TYPE Kilogram : LREAL;
END_TYPE

(* stored: Version 1.1.0.1, ProductVersion 3.1.4024.12
   DUT Kilogram: Id {0e79f689-22d9-4414-a6dd-e72e1f576ede} *)
